FUNCTION_BLOCK ESP32_PIN (* Change pin state *)
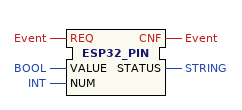
  EVENT_INPUT
    REQ; (* Normal Execution Request *)
  END_EVENT
  EVENT_OUTPUT
    CNF; (* Execution Confirmation *)
  END_EVENT
  VAR_INPUT
    VALUE : BOOL; (* GPIO Value *)
    NUM : INT; (* GPIO Number *)
  END_VAR
  VAR_OUTPUT
    STATUS : STRING; (* Execution Status *)
  END_VAR
END_FUNCTION_BLOCK
